// TwinCAT 3 PLC project tc_project_app
// ProgramVersion: 3.1.4022.2
// libraries:
//   Tc2_EtherCAT, * (Beckhoff Automation GmbH)
//   Tc2_MC2, * (Beckhoff Automation GmbH)
//   Tc2_Standard, * (Beckhoff Automation GmbH)
//   Tc2_System, * (Beckhoff Automation GmbH)
//   Tc2_Utilities, * (Beckhoff Automation GmbH)
//   Tc3_Module, * (Beckhoff Automation GmbH)
// project tree:
//   DUTs/ E_MOTION_MODE.TcDUT, E_OPERATION_MODE.TcDUT, E_OPERATION_MODE_NO.TcDUT, E_PHASING_STATE_MACHINE.TcDUT, E_POSITIONING_STATE_MACHINE.TcDUT, E_VELOCITY_STATE_MACHINE.TcDUT (not stored), ST_AXIS_COMMAND.TcDUT, ST_AXIS_STATUS.TcDUT, ST_CMD_EPICS.TcDUT, ST_STAT_EPICS.TcDUT, ST_INDRADRIVE_IO_INPUT.TcDUT (not stored), ST_INDRADRIVE_IO_OUTPUT.TcDUT, ST_S134_MASTERCONTROLWORD.TcDUT, ST_S135_DRIVESTATUSWORD.TcDUT, ST_S144_SIGNALSTATUSWORD.TcDUT (not stored), ST_S145_SIGNALCONTROLWORD.TcDUT (not stored), TARGET_STATE_MACHINE.TcDUT
//   GVLs/ GVL_ErrorCodes.TcGVL, GVL_Parameters.TcGVL
//   / PlcTask.TcTTO
//   POUs/ MAIN_NORMAL_MOTION.TcPOU (not stored), MAIN.TcPOU
//   POUs/Target/ EL3214.TcPOU, fbIndraDrive.TcPOU, FB_BrakeTorque.TcPOU, FB_ModePhasing.TcPOU, FB_ModeVelo.TcPOU, FB_ModePos.TcPOU, FB_ModeHome.TcPOU, FB_PID.TcPOU, FB_RampVelo.TcPOU, FB_PWM.TcPOU, FB_TargetSuperImpose.TcPOU
//   tc_mca_std_lib/DUTs/ DUT_AxisStatus_v0_01.TcDUT (not stored)
//   tc_mca_std_lib/GVLs/ GVL.TcGVL (not stored)
//   tc_mca_std_lib/POUs/ChangeConfig/ FB_ReadFloatParameter.TcPOU (not stored), FB_ReadParameterInNc_v1_00.TcPOU (not stored), FB_WriteFloatParameter.TcPOU (not stored), FB_WriteParameterInNc_v1_00.TcPOU (not stored)
//   tc_mca_std_lib/POUs/ErrorHandling/ DUT_ErrorState.TcDUT (not stored), DUT_TerminalError.TcDUT (not stored), FB_ErrorList.TcPOU (not stored), FB_TerminalError.TcPOU (not stored), GVL_ErrorSystem.TcGVL (not stored), ST_ErrorSystem.TcDUT (not stored)
//   tc_mca_std_lib/POUs/Hardware/EtherCAT_Terminals/Analog_Inputs/ EL3174_0002.TcPOU (not stored), EL3255.TcPOU (not stored), FB_CalculateFrequency_3702_v0_01.TcPOU (not stored)
//   tc_mca_std_lib/POUs/Hardware/EtherCAT_Terminals/Digital_Inputs/ EL1008.TcPOU (not stored), EL1018.TcPOU (not stored), EL1808.TcPOU (not stored), EL1809.TcPOU (not stored), EL1819.TcPOU (not stored), FB_EL1252ASM_v1_00.TcPOU (not stored)
//   tc_mca_std_lib/POUs/Hardware/EtherCAT_Terminals/Digital_Outputs/ EL2014.TcPOU (not stored), EL2252.TcPOU (not stored), EL2808.TcPOU (not stored), EL2819.TcPOU (not stored)
//   tc_mca_std_lib/POUs/Hardware/EtherCAT_Terminals/Digital_Outputs/External_Types/ dutEL2521_Ctrl.TcDUT (not stored), dutEL2521_Status.TcDUT (not stored)
//   tc_mca_std_lib/POUs/Hardware/EtherCAT_Terminals/Measuring_Terminals/ EL5002.TcPOU (not stored), EL5021.TcPOU (not stored), EL5042.TcPOU (not stored), EL5101.TcPOU (not stored)
//   tc_mca_std_lib/POUs/Hardware/EtherCAT_Terminals/Motion/ EL7211_v1_00.TcPOU (not stored), EL9576_v1_00.TcPOU (not stored)
//   tc_mca_std_lib/POUs/Hardware/EtherCAT_Terminals/System/ EL9410.TcPOU (not stored), EL9505.TcPOU (not stored)
//   tc_mca_std_lib/POUs/Hardware/Other/ EK1200.TcPOU (not stored)
//   tc_mca_std_lib/POUs/Motion/ FB_DriveVirtual.TcPOU (not stored), FB_NcAxis.TcPOU (not stored)
//   tc_mca_std_lib/POUs/Motion/Homing/ FB_HomeDirect.TcPOU (not stored), FB_HomeFinish.TcPOU (not stored), FB_HomePrepare.TcPOU (not stored), FB_HomeReadNcVelocities.TcPOU (not stored), FB_HomeReadSoftLimEnable.TcPOU (not stored), FB_HomeToSwitch.TcPOU (not stored), FB_HomeVirtual.TcPOU (not stored), FB_HomeWriteNcVelocities.TcPOU (not stored), FB_HomeWriteSoftLimEnable.TcPOU (not stored)
//   tc_mca_std_lib/VISUs/ FbDriveVisual.TcVIS (not stored), Visualization.TcVIS (not stored)
// (motion and I/O tree: see PLC project tc_epicscommodule)
// real-time tasks:
//   TASK PlcTaskCom: cycle T#1ms, priority 26, ADS port 350
//   TASK PlcTask: cycle T#1ms, priority 20, ADS port 351

CONFIGURATION tc_project_app
    RESOURCE PLC ON TwinCAT3
        TASK PlcTask(INTERVAL := T#1ms, PRIORITY := 20);
        PROGRAM MAIN WITH PlcTask : MAIN;
    END_RESOURCE
END_CONFIGURATION

// ---- DUTs/E_MOTION_MODE.TcDUT
{attribute 'qualified_only'}
{attribute 'strict'}
TYPE E_MOTION_MODE :
(
	eStop 			:= 0, 
	eJogPositive	:= 1, 
	eJogNegative	:= 2, 
	ePositioning 	:= 3 
);
END_TYPE

// ---- DUTs/E_OPERATION_MODE.TcDUT
{attribute 'qualified_only'}
{attribute 'strict'}
TYPE E_OPERATION_MODE :
(
	eTorqueControl										:= 16#0001,
	eVelocityControl									:= 16#0002,
	ePositionControl_Enc1								:= 16#0003,
	ePositionControl_Enc2								:= 16#0004,
	ePositionControl_Lagless_Enc1						:= 16#000B,
	ePositionControl_Lagless_Enc2						:= 16#000C,
	ePositionControl_DriveControlled_Enc1				:= 16#0103,
	ePositionControl_DriveControlled_Enc2				:= 16#0104,
	ePositionControl_Lagless_Enc1_DriveControlled		:= 16#010B,
	ePositionControl_Lagless_Enc2_DriveControlled		:= 16#010C,
	ePositionControl_DriveControlled_w_AxisControlWord	:= 16#0305,
	ePositionControl_w_AxisControlWord					:= 16#0205,
	eDriveInternal_Interpolation_Enc1					:= 16#0113,
	eDriveInternal_Interpolation_Enc2					:= 16#0114,
	eDriveInternal_Interpolation_Lagless_Enc1			:= 16#011B,
	eDriveInternal_Interpolation_Lagless_Enc2			:= 16#011C,
	eDriveInternal_Interpolation_w_AxisControlWord		:= 16#0315,
	eDriveControlled_Positioning_Enc1					:= 16#0123,
	eDriveControlled_Positioning_Enc2					:= 16#0124,
	eDriveControlled_Positioning_Enc1_Lagless			:= 16#012B,
	eDriveControlled_Positioning_Enc2_Lagless			:= 16#012C,
	eDriveControlled_Positioning_w_AxisControlWord		:= 16#0325,
	ePositioning_BlockModeEnc1							:= 16#0133,
	ePositioning_BlockModeEnc2							:= 16#0134,
	ePositioning_BlockModeLagless_Enc1					:= 16#013B,
	ePositioning_BlockModeLagless_Enc2					:= 16#013C,
	ePositioning_BlockMode_w_AxisControlWord			:= 16#0335,
	eCam_Enc1_VirtualMasterAxis							:= 16#8803,
	eCam_Enc2_VirtualMasterAxis							:= 16#8804,
	eCam_Lagless_Enc1_VirtualMaster_Axis				:= 16#880B,
	eCam_Lagless_Enc2_VirtualMaster_Axis				:= 16#880C,
	eCam_Enc1_RealMasterAxis							:= 16#8813,
	eCam_Enc2_RealMasterAxis							:= 16#8814,
	eCam_Lagless_Enc1_RealMasterAxis					:= 16#881B,
	eCam_Lagless_Enc2_RealMasterAxis					:= 16#881C,
	ePhaseSynch_Enc1_VirtualMasterAxis					:= 16#9003,
	ePhaseSynch_Enc2_VirtualMasterAxis					:= 16#9004,
	ePhaseSynch_Lagless_Enc1_VirtualMasterAxis			:= 16#900B,
	ePhaseSynch_Lagless_Enc2_VirtualMasterAxis			:= 16#900C,
	ePhaseSynch_Enc1_RealMasterAxis						:= 16#9013,
	ePhaseSynch_Enc2_RealMasterAxis						:= 16#9014,
	ePhaseSynch_Lagless_Enc1_RealMasterAxis				:= 16#901B,
	ePhaseSynch_Lagless_Enc2_RealMasterAxis				:= 16#901C,
	eVelocitySynch_VirtualMasterAxis					:= 16#A002,
	eVelocitySynch_RealMasterAxis						:= 16#A012,
	eMotionProfileEnc1_VirtualMasterAxis				:= 16#9803,
	eMotionProfileEnc2_VirtualMasterAxis				:= 16#9804,
	eMotionProfile_Lagless_Enc1_VirtualMasterAxis		:= 16#980B,
	eMotionProfile_Lagless_Enc2_VirtualMasterAxis		:= 16#980C,
	eMotionProfileEnc1_RealMasterAxis					:= 16#9813,
	eMotionProfileEnc2_RealMasterAxis					:= 16#9814,
	eMotionProfile_Lagless_Enc1_RealMasterAxis			:= 16#981B,
	eMotionProfile_Lagless_Enc2_RealMasterAxis			:= 16#981C,
	eVelocity_Synch										:= 16#0142,	
	ePosition_Synch										:= 16#0345
) UINT;
END_TYPE

// ---- DUTs/E_OPERATION_MODE_NO.TcDUT
{attribute 'qualified_only'}
{attribute 'strict'}
TYPE E_OPERATION_MODE_NO :
(
	ePrimaryOpMode 		:= 0, 
	eSecondaryOpMode1 	:= 1, 
	eSecondaryOpMode2 	:= 2, 
	eSecondaryOpMode3 	:= 3, 
	eSecondaryOpMode4 	:= 4, 
	eSecondaryOpMode5 	:= 5, 
	eSecondaryOpMode6 	:= 6, 
	eSecondaryOpMode7 	:= 7	
);
END_TYPE

// ---- DUTs/E_PHASING_STATE_MACHINE.TcDUT
{attribute 'qualified_only'}
{attribute 'strict'}
TYPE E_PHASING_STATE_MACHINE :
(
	POWER_OFF := 0,
	POWER_ON :=1,
	ACCELERATION :=2,
	PHASING :=3
);
END_TYPE

// ---- DUTs/E_POSITIONING_STATE_MACHINE.TcDUT
{attribute 'qualified_only'}
{attribute 'strict'}
TYPE E_POSITIONING_STATE_MACHINE :
(
	POWER_OFF := 0,
	POWER_ON := 1,
	POSITION := 2
);
END_TYPE

// ---- DUTs/ST_AXIS_COMMAND.TcDUT
TYPE ST_AXIS_COMMAND :
STRUCT
	eOperationMode				: E_OPERATION_MODE_NO	:= E_OPERATION_MODE_NO.ePrimaryOpMode;	// (S134.0-2) Defines the Operation mode to use (the different operation modes are configured in the drive) 
	bEnableAxis					: BOOL	:= FALSE; 	// FALSE (S134.13-15): Disable drive 
													// TRUE (S134.13-15): Enable drive (torque on the motor) 
	bHaltAxis					: BOOL	:= FALSE;	// FALSE (S134.13-15): Drive performs a HALT operation (Deceleration of drive while maintaining the max. acceleration (S-0-0138). Requires bEnableAxis to be TRUE) 
													// TRUE (S134.13-15): Drive is not halted
	eMotionMode					: E_MOTION_MODE		:= E_MOTION_MODE.eStop;	// Defines the type of motion that shall be performed. This is not functional in Operation Mode Drive internal interpolation! 
	//bPositioningMode			: BOOL;				// (S346.2&1 FALSE&FALSE): Activates positioning mode according to current Operation mode 
	//bJogPositive				: BOOL;				// (S346.2&1 FALSE&TRUE): Activates jogging in positive direction  
	//bJogNeagtive				: BOOL;				// (S346.2&1 TRUE&FALSE): Activates jogging in negative direction
	//bStopAxis					: BOOL;				// (S346.2&1 TRUE&TRUE): Stops the axis 
	bCommandPositionChange		: BOOL	:= FALSE;	// (S346.5) FALSE: Drive moves to current target position, before positioning to new target position (when bCommandValueAccept is toggled) 
													// (S346.5) TRUE: Immediate of target position, i.e., drive immediately acknowledges the new target position (when bCommandValueAccept is toggled) 
	fCommandPosition			: LREAL	:= 0.0;		// (S47, S258 or S282 according to OperationMode)
	fCommandVelocity			: LREAL	:= 0.0; 	// (S259): The velocity used for Positioning and Jogging
	fCommandAcceleration		: LREAL	:= 0.0;		// (S260): The acceleration used for Positioning and Jogging 
	fCommandDeceleration		: LREAL	:= 0.0;		// (S359): The deceleration used for Positioning and Jogging 
	fFeedrateOverride			: LREAL	:= 100.0; 	// (S108):  Parameter used for variable adjustment of the velocity [0..100%] 
	fTorqueLimit				: LREAL	:= 100.0;	// (S92):  Parameter used for limiting the torque [0..drive/motor limit%] 
	bPositionCommandValue		: BOOL	:= FALSE;	// (S346.3): FALSE: Command position is absolute 
													// (S346.3): TRUE: Command position is relative
	bCommandValueAccept			: BOOL	:= FALSE; 	// (S346.0) Toggle bit (FALSE->TRUE or TRUE->FALSE) to start a positioning command in Operation mode "Drive controlled Positioning"
	bCmd_ErrorReset				: BOOL	:= FALSE;	// (S99): Reset the error of the drive 
	bCmd_SetAbsolutePosition	: BOOL	:= FALSE;	// (P12, C0300): Sets the Absolute position of the drive according to drive configuration 
	bCmd_DriveControlledHoming	: BOOL	:= FALSE;	// (S148, C0600): Starts the homing procedure configured in the drive. NOTE that this does not set the absolute position 
	bCmd_DisableLimits			: BOOL	:= FALSE;	// (bS159, C1300): Disables Monitoring of Position error, Position command error, Velocity error and Acceleration limit
	bCmd_ActivateParameterMode	: BOOL	:= FALSE;	//  (S420, C0400): TRUE: Brings the drive to parameter mode 
	bCmd_ExitParameterMode		: BOOL	:= FALSE;	//  (S422, C0200): TRUE: Brings the drive from parameter mode 
	bCmd_RunVirtualMater		: BOOL	:= FALSE;	//  Jog command to the virtual Master
	fVelocityCommandValue		: LREAL	:= 0.0; 	// (S40): The velocity used for Positioning and Jogging

END_STRUCT
END_TYPE

// ---- DUTs/ST_AXIS_STATUS.TcDUT
TYPE ST_AXIS_STATUS :
STRUCT

	bDriveInParameterMode		: BOOL;		// FALSE (S424): Drive is in Operating mode
											// TRUE (S424): The drive is in parameter mode (parameterization level 1 is active)
	eActualOperationModeNo		: E_OPERATION_MODE_NO	:= E_OPERATION_MODE_NO.ePrimaryOpMode;	// (S134.0-2) Defines the Operation mode to use (the different operation modes are configured in the drive) 
	bDCBusPresent				: BOOL;		// FALSE: DC-bus is not present (drive status bb)
											// TRUE (S135.1&0 TRUE&FALSE): DC-bus present (drive state Ab)
	bAxisEnabled				: BOOL; 	// TRUE (S135.1&0 TRUE&TRUE): Axis is operational with torque (drive state AF)
	bAxisHomedStatus			: BOOL; 	// TRUE (S403.0): Axis absolute position is established 
	bAxisStandStillStatus		: BOOL;		// TRUE (S331): Axis is standing still (velocity below configured threshold) 
	bAxisInTargetPosition		: BOOL;		// TRUE (S437.2): Axis command position is reached
	bAxisConstantVelocityStatus	: BOOL;		// TRUE (S437.4): Axis in constant velocity
	bAxisAccelerationStatus		: BOOL;		// TRUE (S437.5): Axis in acceleration
	bAxisDecelerationStatus		: BOOL;		// TRUE (S437.6): Axis in deceleration
	bAxisJogStatus				: BOOL;		// TRUE (S437.12): Axis in jog mode
	fActualPosition				: LREAL;	// The actual position of the axis
	fActualVelocity				: LREAL;	// The actual velocity of the axis
	fActualTorque				: LREAL;	// The actual torque of the axis
	fPositionError				: LREAL;	// The position error of the axis, i.e. the deviation between the Axis Set position and Actual position
	bCommandChange				: BOOL;		// (S135.5): Bit that toggle every time a new command has been recognised by the drive 
	bCommandValueProcessing		: BOOL;		// FALSE (S115.3): Drive ignores (external) command value input (S47, S258, S282 etc) 
											// TRUE (S115.3): Drive follows (external) command value input (S47, S258, S282 etc) 
	bLimitsDisabled				: BOOL;		// TRUE (S159-C1300): 	Monitoring of Position error, Position command error, Velocity error and Acceleration limit is disabled
											// FALSE (S159-C1300): 	Monitoring of Position error, Position command error, Velocity error and Acceleration limit is enabled 
	bDiagMessage				: BOOL;		// TRUE (S135.11): There is a Diagnostic message on the drive 
	bWarning					: BOOL;		// TRUE (S135.12): There is a warning present on the drive 
	bError 						: BOOL;		// TRUE (S135.13): There is an error present on the drive 
	nDiagMessage				: DWORD;	// (S390) Displays the actual diagnostic message on the drive 
END_STRUCT
END_TYPE

// ---- DUTs/ST_CMD_EPICS.TcDUT
TYPE ST_CMD_EPICS :
STRUCT
	
	bExecute:BOOL:=FALSE;
	bEnable:BOOL:=FALSE;
	bReset:BOOL:=FALSE;
	fVelSet:LREAL:=0;
	fPosSet:LREAL:=0;
	eTargetStateCmd: TARGET_STATE_MACHINE:=0;
	
	//brake
	bBrakeLockOnCmd:BOOL:=FALSE;
	bFreeWheelOnOnCmd:BOOL:=TRUE;
	fBrakeSpNm:LREAL:=0;
END_STRUCT
END_TYPE

// ---- DUTs/ST_STAT_EPICS.TcDUT
TYPE ST_STAT_EPICS :
STRUCT
	
	bError:BOOL:=FALSE;
	nErrorId:UDINT:=0;
	bEnabled:BOOL:=FALSE;
	eTargetState: TARGET_STATE_MACHINE;
    sErrorStr:STRING:='NO ERROR';
	fActTorque:LREAL:=0;
	fActPos:LREAL:=0;
	fActVel:LREAL:=0;	
	fActTemp:LREAL:=0;
	fSetVelRaw:LREAL;
	fBrakeActTemp1:LREAL;
	fBrakeActTemp2:LREAL;
	bBrake1TempAlarm:BOOL;
	bBrake2TempAlarm:BOOL;
END_STRUCT
END_TYPE

// ---- DUTs/ST_INDRADRIVE_IO_OUTPUT.TcDUT
TYPE ST_INDRADRIVE_IO_OUTPUT :	// Contains the data that is sent to the drive
STRUCT
	stS134_MasterControlWord			AT %Q*	: ST_S134_MASTERCONTROLWORD; 	
	nS47_PositionCommandValue			AT %Q*	: DINT; 
	nS258_TargetPosition				AT %Q*	: DINT; 
	nS282_PositioningCommandValue		AT %Q*	: DINT; 
	nS259_PositioningVelocity			AT %Q*	: UDINT; 
	nS260_PositioningAcceleration		AT %Q*	: UDINT; 
	nS359_PositioningDeceleration		AT %Q*	: UDINT; 
	nS108_FeedrateOverride				AT %Q*	: UINT; 
	stS145_SignalControlWord			AT %Q*	: ST_S145_SIGNALCONTROLWORD;
	nS92_BiPolarTorqueLimit				AT %Q*	: INT; 
	nS40_VelocityCommandValue			AT %Q*	: DINT; 

END_STRUCT
END_TYPE

// ---- DUTs/ST_S134_MASTERCONTROLWORD.TcDUT
TYPE ST_S134_MASTERCONTROLWORD :
STRUCT
	{attribute 'hide'}
	bS134_0_CtrlInfo_ServiceCh				: BIT;	// 	Control information for service channel
	{attribute 'hide'}
	bS134_1_CtrlInfo_ServiceCh				: BIT;	// 	Control information for service channel
	{attribute 'hide'}
	bS134_2_CtrlInfo_ServiceCh				: BIT;	// 	Control information for service channel
	{attribute 'hide'}
	bS134_3_CtrlInfo_ServiceCh				: BIT;	// 	Control information for service channel
	{attribute 'hide'}
	bS134_4_CtrlInfo_ServiceCh				: BIT;	// 	Control information for service channel
	{attribute 'hide'}
	bS134_5_CtrlInfo_ServiceCh				: BIT;	// 	Control information for service channel
	{attribute 'hide'}
	bS134_6_RealTime_Bit1					: BIT;	// 	Real time bit1
	{attribute 'hide'}
	bS134_7_RealTime_Bit2					: BIT;	// 	Real time bit2
	bS134_CmdOperationMode_Bit0				: BIT;	// 	(bS134_CmdOpMode_B2 | bS134_CmdOpMode_B2 | bS134_CmdOpMode_B0)
													//	000: Primary mode of operation
													// 	001: Secondary operation mode 1
													// 	010: Secondary operation mode 2, etc
	bS134_CmdOperationMode_Bit1				: BIT;	// 	(bS134_CmdOpMode_B2 | bS134_CmdOpMode_B2 | bS134_CmdOpMode_B0)
													//	000: Primary mode of operation
													// 	001: Secondary operation mode 1
													// 	010: Secondary operation mode 2, etc
	bS134_IPOSYNC							: BIT;	// 	Interpolator clock, toggles when new command values are to be transmitted 
	bS134_CmdOperationMode_Bit2				: BIT;	// 	(bS134_CmdOpMode_B2 | bS134_CmdOpMode_B2 | bS134_CmdOpMode_B0)
													//	000: Primary mode of operation
													// 	001: Secondary operation mode 1
													// 	010: Secondary operation mode 2, etc
	{attribute 'hide'}
	bS134_12_Reserved						: BIT;	// 	Reserved
	bS134_DriveHalt							: BIT;	// 	1-0 change: deceleration of drive while maintaining the max. acceleration (S-0-0138) 
													//	(only possible when bit bS134_DriveEnable and bS134_DriveOn = TRUE)
	bS134_DriveEnable						: BIT;	// 	TRUE -> FALSE transition: torque disable without delay (independent of bit bS134_DriveOn or bS134_DriveHalt)
	bS134_DriveOn							: BIT;	// 	TRUE -> FALSE transition: best possible deceleration (only possible if bit bS134_DriveEnable = TRUE)


	

	


END_STRUCT
END_TYPE

// ---- DUTs/ST_S135_DRIVESTATUSWORD.TcDUT
TYPE ST_S135_DRIVESTATUSWORD :
STRUCT
	{attribute 'hide'}
	bS135_0_CtrlInfo_ServiceCh				: BIT;	// 	Control information for service channel
	{attribute 'hide'}
	bS135_1_CtrlInfo_ServiceCh				: BIT;	// 	Control information for service channel
	{attribute 'hide'}
	bS135_2_CtrlInfo_ServiceCh				: BIT;	// 	Control information for service channel
	{attribute 'hide'}
	bS135_3_CmdValProcessingStatus			: BIT;	// 	Status of command value processing
	{attribute 'hide'}
	bS135_4_Reserved						: BIT;	// 	Reserved
	bS135_CommandChange 					: BIT;	// 	Toggling bit to acknowledge that the Command status has changed 
	{attribute 'hide'}
	bS135_6_RealTime_Bit1					: BIT;	// 	Real time bit1
	{attribute 'hide'}
	bS135_7_RealTime_Bit2					: BIT;	// 	Real time bit2
	bS135_ActualOperationMode_Bit0			: BIT;	// 	(bS135_ActOpMode_B2 | bS135_ActOpMode_B2 | bS135_ActOpMode_B0)
													//	000: Primary operation mode active
													// 	001: Secondary operation mode 1 active
													// 	010: Secondary operation mode 2 active, etc
	bS135_ActualOperationMode_Bit1			: BIT;	// 	(bS135_ActOpMode_B2 | bS135_ActOpMode_B2 | bS135_ActOpMode_B0)
													//	000: Primary operation mode active
													// 	001: Secondary operation mode 1 active
													// 	010: Secondary operation mode 2 active, etc
	bS135_ActualOperationMode_Bit2			: BIT;	// 	(bS135_ActOpMode_B2 | bS135_ActOpMode_B2 | bS135_ActOpMode_B0)
													//	000: Primary operation mode active
													// 	001: Secondary operation mode 1 active
													// 	010: Secondary operation mode 2 active, etc
	bS135_Class3_Diag_Mess					: BIT;	// 	TRUE: There is a Class 3 Diagnostic message present in the drive
	bS135_Class2_Diag_Warn					: BIT;	// 	TRUE: There is a Warning present in the drive
	bS135_Class1_Diag_Err					: BIT;	// 	TRUE: There is a Error present in the drive
	bS135_ReadyForOperation_Bit0			: BIT;	// 	(bS135_ReadyForOp_B1 | bS135_ReadyForOp_B0)
													//	00: Not ready for power on (e.g. drive in "P2")
													//	01: Ready for power on ("bb") (A0013)
													//	10: Control section and power section ready for op. ("Ab") (A0012)
													//	11: In operation, with torque (e.g. "AF")
	bS135_ReadyForOperation_Bit1			: BIT;	// 	(bS135_ReadyForOp_B1 | bS135_ReadyForOp_B0)
													//	00: Not ready for power on (e.g. drive in "P2")
													//	01: Ready for power on ("bb") (A0013)
													//	10: Control section and power section ready for op. ("Ab") (A0012)
													//	11: In operation, with torque (e.g. "AF")

	


	


END_STRUCT
END_TYPE

// ---- DUTs/TARGET_STATE_MACHINE.TcDUT
{attribute 'qualified_only'}
{attribute 'strict'}
TYPE TARGET_STATE_MACHINE :
(
	POWER_OFF := 0,
	POWER_ON := 1,
	CONSTANT_VELOCITY :=2,
	POSITIONING :=3,
	PHASING :=4,
	HOMING := 5
	
	
	
);
END_TYPE

// ---- GVLs/GVL_ErrorCodes.TcGVL
{attribute 'qualified_only'}
VAR_GLOBAL
	nErrorCodeOKId:UDINT:=0;
	nErrorCodeOKStr:STRING:='NO ERROR';
	nErrorNoLatchId:UDINT:=1000;
	sErrorNoLatchStr:STRING:='NO LATCH FROM DRIVE';
END_VAR

// ---- GVLs/GVL_Parameters.TcGVL
{attribute 'qualified_only'}
VAR_GLOBAL
	fSpeedToleranceRpm: LREAL := 0.05;
END_VAR

VAR_GLOBAL CONSTANT
	nSectors: LREAL :=36;
    nPulseFreqHz:LREAL:=14;
	fNominalSpeedRpm: LREAL := GVL_Parameters.nPulseFreqHz/GVL_Parameters.nSectors*60;
	fNominalSpeedAdjust: LREAL:=0.001;//-0.0002;  //Timing system vs drive clock tuning. Automize later!
	fPhaseSpeedTol:LREAL:=0.02;   //Speed for last rev needs to be below before start to phase
	fHomeSpeedRpm: LREAL := 1;
    fMaximumSPeedRpm: LREAL := GVL_Parameters.fNominalSpeedRpm*1.1;
	nMaxMotorTemperature: INT:= 80;
	nMaxBrakeTemperature: INT:= 100;
	fWheelDiameter:LREAL:=2500;
	fAccDefault:LREAL:=0.039;  //RPM/S^2 (0.039 => tn min to 23.3) 
	nPhaseErrorFilterSize:INT:=36;  //Two revs
	nVeloInRangeCount:INT:=100;
	nSuperPosMaxCyclesToOutput:INT:=100;
	fSuperPosDutyCycle:LREAL:=2.0/3.0;
	nTaskSampleTime:INT:=1;
	nPhasePIDReducedSampleRateFactor:INT:=1;   //run pid every time new pulse
END_VAR

// ---- POUs/MAIN.TcPOU
PROGRAM MAIN
VAR
	stAmsNetId	AT %I*	              : AMSNETID;
	nPort	AT %I*                    : WORD;
	nMasterAxisPosition AT %I*        : DINT;
	nAdditivePositionSetpoiunt AT %Q* : DINT;
	nAdditiveTorqueSetpoint    AT %Q* : INT;   // Unit 0.1%  (10=1%)
	dLatchedPosition AT %I*           : DINT;
	iBrakeSpRaw AT %Q*                : INT := 0;
	//iRotMotorTempRaw AT %I*           : INT := 0;
    fbTemp                            : EL3214;
	bBrakeFreewheelOn AT %Q*          : BOOL;
	bBrakeLockedOn AT %Q*             : BOOL;
    inputDummy AT %I*                 : BOOL;
	inputDigSens1 AT %I*              : BOOL;
	inputDigSens2 AT %I*              : BOOL;
	fbBrakeTorque                     : FB_BrakeTorque;  // Control brake
	fbModePhase                       : FB_ModePhasing;	 // Phasing Mode
	fbRampVelo                        : FB_RampVelo;
	fbModeVelo                        : FB_ModeVelo;     // Velocity Mode
	fbModePos                         : FB_ModePos;      // Positioning Mode
	fbModeHome                        : FB_ModeHome;     // Homing Mode
	fbIndraDrive                      : fbIndraDrive;    // Control of drive
	stStatEpics                       : ST_STAT_EPICS;   // Status to EPICS
	stCmdEpics                        : ST_CMD_EPICS;    // Control to EPICS 
	stCommands                        : ST_AXIS_COMMAND; // Control to drive
	stStatus                          : ST_AXIS_STATUS;  // Status from drive
	eTargetStateOld                   : TARGET_STATE_MACHINE;
	addStartupTorqueTrigger           : BOOL:=FALSE;
	iTorqueCommandValue  AT %Q*       : INT := 0;
END_VAR

// Monitor temperature
ACT_Temperature();
// Control brake
ACT_Brake();


// Enable Axis independent of state
stCommands.bEnableAxis :=stCmdEpics.bEnable;
stCommands.bHaltAxis:=stCmdEpics.bExecute;
stStatEpics.bEnabled:=stStatus.bAxisEnabled;
stCommands.bCmd_ErrorReset:=stCmdEpics.bReset;

IF NOT stCmdEpics.bEnable THEN
  stCmdEpics.bExecute:=FALSE;
END_IF

stCommands.fCommandAcceleration:=GVL_Parameters.fAccDefault;
stCommands.fCommandDeceleration:=GVL_Parameters.fAccDefault;
stCommands.bCmd_DriveControlledHoming:=FALSE;

// Only allow state change if execute is low
IF stCmdEpics.eTargetStateCmd <> stStatEpics.eTargetState AND NOT stCmdEpics.bexecute THEN
	stStatEpics.eTargetState:=stCmdEpics.eTargetStateCmd;
END_IF

//nAdditiveTorqueSetpoint:=0;
//IF NOT  stCmdEpics.bExecute THEN
//	addStartupTorqueTrigger:=TRUE;
//END_IF

CASE stStatEpics.eTargetState OF 
	TARGET_STATE_MACHINE.CONSTANT_VELOCITY:
		fbModeVelo(
            bExecute:=         stCmdEpics.bExecute,
            bReset:=           stCmdEpics.bReset,
			fVelSet:=          stCmdEpics.fVelSet,
			stStatus:=	       stStatus,	
			stCommands:=       stCommands);
			
			//ramp velocity with selected acceleration
			fbRampVelo(bExecute:=stCmdEpics.bExecute,
              fVelSetIn:=fbModeVelo.fSpeedSetpoint,
              iBlockSampleTimeMicroS:=GVL_Parameters.nTaskSampleTime*1000,
              fVelSetOut:=stCommands.fVelocityCommandValue,
              fVelActIn:=stStatus.fActualVelocity/10);
			  
// add extra torque att startup TEST
		//	IF stStatus.bAxisEnabled AND stCmdEpics.bExecute AND stCmdEpics.fVelSet > 0 THEN
		//		IF stStatus.fActualVelocity/10< stCmdEpics.fVelSet/2 THEN
		//	        nAdditiveTorqueSetpoint:=100;  //Add 10% when under x rpm
		//		ELSIF stStatus.fActualVelocity/10 > stCmdEpics.fVelSet/2 THEN
		//			nAdditiveTorqueSetpoint:=40;
		//		END_IF
		//	END_IF

			
	TARGET_STATE_MACHINE.POSITIONING:
		fbModePos(
            bExecute:=         stCmdEpics.bExecute,
            bReset:=           stCmdEpics.bReset,
			fVelSet:=          stCmdEpics.fVelSet,
			fPosSet:=          stCmdEpics.fPosSet,
			stStatus:=         stStatus,	
			stCommands:=       stCommands);
		
	TARGET_STATE_MACHINE.PHASING:
   		fbModePhase(
			bExecute:=         stCmdEpics.bExecute,
            bReset:=           stCmdEpics.bReset,
			stStatus:=	       stStatus,
			dLatchedPosition:= dLatchedPosition,
			ePhaseType:=stCmdEpics.ePhaseCntrlAlg,
			stCommands:=       stCommands);
			
			//ramp velocity with selected acceleration (as long as not phasing)
			IF NOT fbModePhase.bPhasing THEN
              fbRampVelo(bExecute:=stCmdEpics.bExecute,
                fVelSetIn:=fbModePhase.fSpeedSetpoint,
                iBlockSampleTimeMicroS:=GVL_Parameters.nTaskSampleTime*1000,
                fVelSetOut:=stCommands.fVelocityCommandValue,
                fVelActIn:=fbModePhase.fLastSectorVelocity);
			ELSE // if phasing then take setpoint direct from fbModePhase
			  stCommands.fVelocityCommandValue:=fbModePhase.fSpeedSetpoint;
            END_IF
						
	TARGET_STATE_MACHINE.HOMING:
        fbModeHome( 
            bExecute:=         stCmdEpics.bExecute,
            bReset:=           stCmdEpics.bReset,
			fVelSet:=          stCmdEpics.fVelSet,
			fPosSet:=          stCmdEpics.fPosSet,
			stStatus:=	       stStatus,	
			stCommands:=       stCommands);
			
	TARGET_STATE_MACHINE.TORQUE:
		stCommands.eOperationMode:=E_OPERATION_MODE_NO.eSecondaryOpMode7;
	    stCommands.eMotionMode :=e_Motion_mode.eJogPositive;
	
	  ELSE  // No valid state
		  
		stCmdEpics.bExecute:=FALSE;
        stCmdEpics.bEnable:=FALSE;
		stCommands.fVelocityCommandValue:=0;
		stCommands.fCommandVelocity:=0;
		
END_CASE

IF NOT stCmdEpics.bExecute THEN
	stCommands.fVelocityCommandValue:=0;
END_IF

// TODO: Why I put this here?
stCommands.eMotionMode:=E_MOTION_MODE.eStop;

// Rexroth FB
fbIndraDrive(
	AmsNetId:= stAmsNetId, 
	AdsAddr_Port:= nPort, 
	stAxisCommands:= stCommands, 
	stDriveStatus:= , 
	stAxisStatus=> stStatus, 
	stDriveCommands=> );

// Calculate values for status in EPICS
stStatEpics.fSetVelRaw:= DINT_TO_LREAL(MAIN.fbIndraDrive.stDriveCommands.nS40_VelocityCommandValue)/10000;	
stStatEpics.fActPos:=stStatus.fActualPosition;
stStatEpics.fActTorque:=stStatus.fActualTorque;
stStatEpics.fActVel:=stStatus.fActualVelocity/10;

// Error handling
ACT_Error();

eTargetStateOld:=stStatEpics.eTargetState;

ACTION ACT_Brake:
// Function: Control of brake for simulation of traction
// Use at target test rig
// Author: Anders Sandström 2019

bBrakeFreewheelOn:=stCmdEpics.bFreeWheelOnOnCmd;
bBrakeLockedOn:=stCmdEpics.bBrakeLockOnCmd;

fbBrakeTorque(iTorqueValueinNm:=stCmdEpics.fBrakeSpNm);
iBrakeSpRaw:=fbBrakeTorque.iTorqueScaled;
END_ACTION

ACTION ACT_Diag:
// Function: Some parameters just for debugging
// Note: Do not need to be executed, can be watched online anyway..
// Author: Anders Sandström 2019

	stCommands.bCmd_ActivateParameterMode;//True puts the drive in parameter mode
	stCommands.bCmd_DisableLimits;// True disables monitoring of errors
	stCommands.bCmd_DriveControlledHoming;// True starts homing procedure defined in the drive
	stCommands.bCmd_ErrorReset;
	stCommands.bCmd_ExitParameterMode;
	stCommands.bCmd_RunVirtualMater;// Jog command to the virtual master
	stCommands.bCmd_SetAbsolutePosition;
	stCommands.bCommandPositionChange;// Drive moves to the current target position, when bCommandVAlueAccept toggled, drive moves to the new target position
	stCommands.bCommandValueAccept;// Used in "Drive positioning Mode" to update the target position when toggled
	stCommands.bEnableAxis;
	stCommands.bHaltAxis;// Performs halt on the drive, bEnableaxis has to be TRUE
	stCommands.bPositionCommandValue;//0=Absolute;1=Relative
	stCommands.eMotionMode;
	stCommands.eOperationMode;
	stCommands.fCommandAcceleration;// Acceleration used for positioning and jogging
	stCommands.fCommandDeceleration;// Deceleration used for positioning and jogging
	stCommands.fCommandPosition;
	stCommands.fCommandVelocity;// Velocity used for positioning and jogging
	stCommands.fFeedrateOverride;// Parameter used for adjustment of the velocity (0,100)%
	stCommands.fTorqueLimit;
	stCommands.fVelocityCommandValue;// S40, velocity used for positining and jogging (in velocity mode)
	stStatus.bAxisEnabled;
END_ACTION

ACTION ACT_Error:
// Function: Error handling
// Author: Anders Sandström 2019

IF stStatEpics.eTargetState = TARGET_STATE_MACHINE.PHASING THEN
  IF fbModePhase.bError AND NOT stStatEpics.bError THEN
	  stStatEpics.bError:=fbModePhase.bError;
	  stStatEpics.nErrorId:=fbModePhase.nErrorId;
	  stStatEpics.sErrorStr:=fbModePhase.sErrorStr;
  END_IF
  
ELSIF stStatEpics.eTargetState = TARGET_STATE_MACHINE.CONSTANT_VELOCITY THEN
   IF fbModeVelo.bError AND NOT stStatEpics.bError THEN
	  stStatEpics.bError:=fbModeVelo.bError;
	  stStatEpics.nErrorId:=fbModeVelo.nErrorId;
	  stStatEpics.sErrorStr:=fbModeVelo.sErrorStr;
  END_IF
  
ELSIF stStatEpics.eTargetState = TARGET_STATE_MACHINE.POSITIONING THEN
  IF fbModePos.bError AND NOT stStatEpics.bError THEN
	  stStatEpics.bError:=fbModePos.bError;
	  stStatEpics.nErrorId:=fbModePos.nErrorId;
	  stStatEpics.sErrorStr:=fbModePos.sErrorStr;
  END_IF
  
ELSIF stStatEpics.eTargetState = TARGET_STATE_MACHINE.HOMING THEN
  IF fbModeHome.bError AND NOT stStatEpics.bError THEN
	  stStatEpics.bError:=fbModeHome.bError;
	  stStatEpics.nErrorId:=fbModeHome.nErrorId;
	  stStatEpics.sErrorStr:=fbModeHome.sErrorStr;
  END_IF
  
END_IF


IF stcmdEpics.bReset THEN
	stStatEpics.bError:=FALSE;
	stStatEpics.nErrorId:=GVL_ErrorCodes.nErrorCodeOKId;
	stStatEpics.sErrorStr:=GVL_ErrorCodes.nErrorCodeOKStr;
	stStatEpics.bBrake1TempAlarm:=FALSE;
	stStatEpics.bBrake2TempAlarm:=FALSE;
END_IF
END_ACTION

ACTION ACT_Temperature:
// Function: Monitor tempertures
// Interlock motion on temperatures
// Author: Anders Sandström 2019

fbTemp(En:=TRUE);

IF fbTemp.bError THEN
	stCmdEpics.bExecute:=0;
	stCmdEpics.bEnable:=0;
END_IF

stStatEpics.fActTemp:=fbTemp.iAi_Ch1_Value/10.0;
stStatEpics.fBrakeActTemp1:=fbTemp.iAi_Ch2_Value/10.0;
stStatEpics.fBrakeActTemp2:=fbTemp.iAi_Ch3_Value/10.0;

// Motor Temperature Monitoring Interlock
IF (stStatEpics.fActTemp >= GVL_Parameters.nMaxMotorTemperature)  OR fbTemp.iAi_Ch1_Stat >0 THEN
	stCmdEpics.bEnable:= FALSE;
	stCmdEpics.bExecute:= FALSE;	
END_IF

//Brake temperature monitoring Interlock 1
IF (stStatEpics.fBrakeActTemp1 >= GVL_Parameters.nMaxBrakeTemperature) OR fbTemp.iAi_Ch2_Stat >0 OR stStatEpics.bBrake1TempAlarm THEN
	stCmdEpics.bEnable:= FALSE;
	stCmdEpics.bExecute:= FALSE;		
    stStatEpics.bBrake1TempAlarm:=TRUE; 
END_IF
//Brake temperature monitoring Interlock 2
IF (stStatEpics.fBrakeActTemp2 >= GVL_Parameters.nMaxBrakeTemperature) OR fbTemp.iAi_Ch3_Stat >0 OR stStatEpics.bBrake2TempAlarm THEN
	stCmdEpics.bEnable:= FALSE;
	stCmdEpics.bExecute:= FALSE;		
    stStatEpics.bBrake2TempAlarm:=TRUE; 
END_IF
END_ACTION

END_PROGRAM

// ---- POUs/Target/EL3214.TcPOU
//EL3214 | 4-channel analog input terminal, PT100 (RTD)
FUNCTION_BLOCK EL3214

VAR_INPUT
	En: BOOL;
	iTerminal_ID : INT;
END_VAR

VAR_OUTPUT
	EnO: BOOL;
	iAi_Ch1_Value : INT;
	iAi_Ch2_Value : INT;
	iAi_Ch3_Value : INT;
	iAi_Ch4_Value : INT;
	iAi_Ch1_Stat : BYTE;
	iAi_Ch2_Stat : BYTE;
	iAi_Ch3_Stat : BYTE;
	iAi_Ch4_Stat : BYTE;
	bError: BOOL;
END_VAR

VAR
	//Channels
	AI_RTD_Ch_1_Status	AT %I* : WORD;
	AI_RTD_Ch_1_Value 	AT %I* : INT;
	AI_RTD_Ch_2_Status 	AT %I* : WORD;
	AI_RTD_Ch_2_Value 	AT %I* : INT;
	AI_RTD_Ch_3_Status 	AT %I* : WORD;
	AI_RTD_Ch_3_Value 	AT %I* : INT;
	AI_RTD_Ch_4_Status 	AT %I* : WORD;
	AI_RTD_Ch_4_Value 	AT %I* : INT;
	
	//Terminal status
	WcState_WcState AT %I*: BOOL;
	InfoData_State AT %I*: UINT;
END_VAR

(*
* TODO:
* Status words of the channels
*)

EnO := En;

IF En THEN
	iAi_Ch1_Stat:=WORD_TO_BYTE(AI_RTD_Ch_1_Status);
	iAi_Ch2_Stat:=WORD_TO_BYTE(AI_RTD_Ch_2_Status);
	iAi_Ch3_Stat:=WORD_TO_BYTE(AI_RTD_Ch_3_Status);
	iAi_Ch4_Stat:=WORD_TO_BYTE(AI_RTD_Ch_4_Status);
	
    bError:=WcState_WcState OR NOT (InfoData_State=8);
 
	IF bError = FALSE THEN
		iAi_Ch1_Value := AI_RTD_Ch_1_Value;
		iAi_Ch2_Value := AI_RTD_Ch_2_Value;
		iAi_Ch3_Value := AI_RTD_Ch_3_Value;
		iAi_Ch4_Value := AI_RTD_Ch_4_Value;
	ELSE
		iAi_Ch1_Value := 32768;
		iAi_Ch2_Value := 32768;
		iAi_Ch3_Value := 32768;
		iAi_Ch4_Value := 32768;
	END_IF
END_IF

END_FUNCTION_BLOCK

// ---- POUs/Target/FB_BrakeTorque.TcPOU
FUNCTION_BLOCK FB_BrakeTorque
VAR_INPUT
	iTorqueValueinNm: LREAL;
END_VAR
VAR_OUTPUT
	iTorqueScaled: INT; //Scaled torque value 
END_VAR
VAR
	iTorqueMin:LREAL := 2; // Min brake torque in Nm
	iTorqueMax:LREAL := 200; // Max brake torque in Nm
	iVoltageDecMin:INT := 0; // 0V in decimal representation
	iVoltageDecMax:INT := 32767; //10V in decimal representation
END_VAR

// Function: Interface to brake eon target test rig
// Author: Anders Sandström 2018

IF iTorqueValueinNm >=2 THEN	
  iTorqueScaled := LREAL_TO_INT(((iTorqueValueinNm-iTorqueMin)/(iTorqueMax-iTorqueMin))*(iVoltageDecMax-iVoltageDecMin) + iVoltageDecMin);
ELSE
  iTorqueScaled:=0;
END_IF

END_FUNCTION_BLOCK

// ---- POUs/Target/FB_ModePhasing.TcPOU
FUNCTION_BLOCK FB_ModePhasing
VAR_INPUT
	bExecute:BOOL;
	bReset: BOOL;
	stStatus: ST_AXIS_STATUS;
    dLatchedPosition: DINT;
	fPhaseOffsetDeg: LREAL;
    fPhaseControlKp: LREAL := 0.00001;
	///Ti
	fPhaseControlTn: LREAL := 0;
	///Td
	fPhaseControlTv: LREAL := 0;
	///derviative damping
	fPhaseControlTd: LREAL := 0;
	bPhaseControlReset: BOOL := FALSE;
	
	// for own pid (use kp above)
	fPhaseControlKi: LREAL := 0.0001;
	fPhaseControlKd: LREAL := 0.0001;
	fPhaseControlKff: LREAL := 0.0;
END_VAR
VAR_OUTPUT
	bError: BOOL;
	nErrorId: UDINT;
	sErrorStr: STRING:=GVL_ErrorCodes.nErrorCodeOKStr;
	bPhasing:BOOL;
	fSpeedSetpoint: LREAL;
	fCtrlOutput:LREAL;
END_VAR
VAR_IN_OUT
	stCommands: ST_AXIS_COMMAND;
END_VAR
VAR
	fLatchedPositionOld: LREAL;
	fDistBetweenLastPulses: LREAL;
	fLastSectorVelocity: LREAL;
	fVelocityFromDriveScaled: LREAL;
	fClosestSectorId: LREAL;
	nClosestSectorId: INT;
	fLatchedPosition:LREAL;
	//fbPhasePID: Tc2_Utilities.FB_BasicPID;
	fbPhasePID: FB_PID;
	fPhaseError: LREAL;
	fPhaseErrorFiltered:LREAL;
	fPhaseErrorMM: LREAL:=0;
	dLatchedPositionOld:DINT;
	fPhaseErrorAcc:LREAL;
	ii: INT;
	bTestReset: BOOL;
	bNewTriggPulse:BOOL:=FALSE;
	fArrayFiltVelo: ARRAY[ 0 ..35] OF LREAL;
	fArrayPhaseErrorFilt: ARRAY[ 0 ..99] OF LREAL;
	fArrayPhaseErrorLongTime: ARRAY[ 0 ..99] OF LREAL;
	iFiltVeloArrayIndex:INT:=0;
	fLastSectorVelocityOld:LREAL:=0;
	i:INT:=0;
	fMaxValue:LREAL:=0;
	fMinValue:LREAL:=0;
	fRange:LREAL:=0;
	iRangeOKCounter:INT:=0;
	iRangeOKCounterOld:INT:=0;
	nChoosenSector:INT:=0;
	bPhaseAlgTrigg: BOOL;
	fbPWM: FB_PWM;
	fbSuperImpose:FB_TargetSuperImpose;
	bExecuteSuperImpose: BOOL;
	fPhaseErrorSlope: LREAL;
	iNominalVelCounter:INT:=0;
	fDeltaVelo: LREAL;
	bVeloStable:BOOL:=FALSE;
	timerCheckLatchFreq:TON;
	fNomSpeedSetAdjust: LREAL := 0;
	bTEst: BOOL := FALSE;
	fPidAdd: LREAL := 0;
	fCtrlCycleTime: INT;
	fTn: INT;
END_VAR

// Function: 
// 1. Wait for stable velocity then start "phasing" 
// 2. Choose sector for control
// 3. Calculate phase error (buffer several revs and filter)
// 4. Adjust velo setpoint to minimize phase error
// Author: Anders Sandström 2018

stCommands.fCommandDeceleration:=GVL_Parameters.fAccDefault;	
stCommands.fCommandAcceleration:= GVL_Parameters.fAccDefault;
stCommands.eMotionMode :=e_Motion_mode.eJogPositive;
stCommands.eOperationMode:=e_Operation_mode_no.eSecondaryOpMode2;
fVelocityFromDriveScaled:=stStatus.fActualVelocity/10;
bNewTriggPulse:=FALSE;
bPhasing:=FALSE;
fNomSpeedSetAdjust:=GVL_Parameters.fNominalSpeedRpm + GVL_Parameters.fNominalSpeedAdjust; // Adjust speed setpoint
bPhasing:=bPhaseAlgTrigg;

// Reset alg
IF NOT bExecute OR bPhaseControlReset THEN
 bPhaseAlgTrigg:=FALSE;
END_IF

fLatchedPositionOld:=fLatchedPosition;
fLatchedPosition:=DINT_TO_LREAL(dLatchedPosition)/10000.0;

// New trigger from timing system
IF (fLatchedPosition-fLatchedPositionOld)<>0 THEN
  IF(fLatchedPositionOld>fLatchedPosition) THEN
	fDistBetweenLastPulses:=(360-fLatchedPositionOld+fLatchedPosition);
  ELSE
	fDistBetweenLastPulses:=fLatchedPosition-fLatchedPositionOld;
  END_IF
  bNewTriggPulse:=TRUE;
  fLastSectorVelocity:=fDistBetweenLastPulses*GVL_Parameters.nPulseFreqHz*60/360;
  nClosestSectorId:= LREAL_TO_INT(fLatchedPosition/10);
  
  // Check if stable velocity (close to nominal)	
  iRangeOKCounterOld:=iRangeOKCounter;
  fArrayFiltVelo[iFiltVeloArrayIndex]:=fLastSectorVelocity;
  iFiltVeloArrayIndex:=iFiltVeloArrayIndex+1;
  IF iFiltVeloArrayIndex>35 THEN
	iFiltVeloArrayIndex:=0;
  END_IF
  fLastSectorVelocityOld:=fLastSectorVelocity;
  fMaxValue:=fArrayFiltVelo[0];
  fMinValue:=fArrayFiltVelo[0];
  FOR i:=1 TO 35 BY 1 DO
     IF fArrayFiltVelo[i]> fMaxValue THEN
	   fMaxValue:=fArrayFiltVelo[i];  
     END_IF
     IF fArrayFiltVelo[i]< fMinValue THEN
	   fMinValue:=fArrayFiltVelo[i];  
     END_IF
  END_FOR;
  fRange:=fMaxValue-fMinValue;
  IF fRange < GVL_Parameters.fPhaseSpeedTol AND 
     ABS(fNomSpeedSetAdjust-fMinValue) < GVL_Parameters.fPhaseSpeedTol AND  
     ABS(fNomSpeedSetAdjust-fMaxValue) < GVL_Parameters.fPhaseSpeedTol THEN
	IF iRangeOKCounter <= GVL_Parameters.nVeloInRangeCount THEN
      iRangeOKCounter:=iRangeOKCounter+1;
	END_IF
  ELSE
	iRangeOKCounter:=0; 
  END_IF
  bVeloStable:=iRangeOKCounter >= GVL_Parameters.nVeloInRangeCount;
  IF bVeloStable AND NOT bPhaseAlgTrigg (*AND bTEst*) THEN
    nChoosenSector:=nClosestSectorId-1;
    bPhaseAlgTrigg:=TRUE;
    MEMSET(destAddr:=ADR(fArrayPhaseErrorFilt[0]),0,SIZEOF(fArrayPhaseErrorFilt));
    fPhaseErrorFiltered:=0;
  END_IF
END_IF

//Ensure that pulses arrive from timing system when velocity is above certain limit
timerCheckLatchFreq(IN:=fLatchedPosition = fLatchedPositionOld AND ABS(stStatus.fActualVelocity)>0,PT:=LREAL_TO_TIME(1000/GVL_Parameters.nPulseFreqHz*2));

IF NOT bPhaseAlgTrigg THEN
  fPhaseError:=nClosestSectorId*10-fLatchedPosition;
END_IF

IF bNewTriggPulse THEN
  nChoosenSector:=nChoosenSector+1;
  IF nChoosenSector > 35 THEN
    nChoosenSector:=0;
  END_IF	
END_IF

// Calculate phase error
IF bPhaseAlgTrigg THEN
  fPhaseError:=nChoosenSector*10-fLatchedPosition;
  IF fPhaseError >=180 THEN
	fPhaseError:=360-fPhaseError;
  ELSIF fPhaseError<-180 THEN
	fPhaseError:=fPhaseError+360;
  END_IF
ELSE
  fPhaseError:=nClosestSectorId*10-fLatchedPosition;
END_IF
fPhaseErrorMM:=fPhaseError*GVL_Parameters.fWheelDiameter*pi/360.0; 

//Filter phase error
IF bNewTriggPulse THEN
	MEMMOVE(destAddr:=ADR(fArrayPhaseErrorFilt[1]),srcAddr:=ADR(fArrayPhaseErrorFilt[0]),SIZEOF(LREAL)*(GVL_Parameters.nPhaseErrorFilterSize-1));
	fArrayPhaseErrorFilt[0]:=fPhaseErrorMM;
	fPhaseErrorFiltered:=0;
	FOR ii := 0 TO (GVL_Parameters.nPhaseErrorFilterSize-1) DO
		fPhaseErrorFiltered:=fPhaseErrorFiltered+fArrayPhaseErrorFilt[ii];
	END_FOR
	fPhaseErrorFiltered:=fPhaseErrorFiltered/GVL_Parameters.nPhaseErrorFilterSize;
END_IF

IF NOT fbSuperImpose.bBusy  THEN
  bExecuteSuperImpose:= NOT bExecuteSuperImpose;
END_IF

//Drops very fast from positive to negative error. So, Adjust more gently when phase error is positive
IF(fPhaseErrorFiltered > 0) THEN  //Pos error
  IF ABS(fPhaseErrorFiltered)>10 THEN
    fDeltaVelo:= 0.003;
  ELSIF ABS(fPhaseErrorFiltered)>4 THEN
    fDeltaVelo:= 0.0025;
  ELSIF ABS(fPhaseErrorFiltered)>1 THEN
    fDeltaVelo:= 0.002;
  ELSIF ABS(fPhaseErrorFiltered)>0.5 THEN
    fDeltaVelo:= 0.0015;
  ELSE
	fDeltaVelo:= 0.0015;
  END_IF
ELSE // neg error
  IF ABS(fPhaseErrorFiltered)>10 THEN  
    fDeltaVelo:= 0.003;
  ELSIF ABS(fPhaseErrorFiltered)>4 THEN
    fDeltaVelo:= 0.0025;
  ELSIF ABS(fPhaseErrorFiltered)>1 THEN
    fDeltaVelo:= 0.002;
  ELSIF ABS(fPhaseErrorFiltered)>0.5 THEN
    fDeltaVelo:= 0.0015;
  ELSE
	fDeltaVelo:= 0.0015;
  END_IF	
END_IF

//Adjust nominal speed (this function should be automated (adaptive))
fSpeedSetpoint:=fNomSpeedSetAdjust;
IF fSpeedSetpoint>GVL_Parameters.fMaximumSPeedRpm THEN
  fSpeedSetpoint:=GVL_Parameters.fMaximumSPeedRpm; 
END_IF
IF NOT bExecute THEN
  fSpeedSetpoint:=0;	
END_IF
IF bNewTriggPulse AND bPhaseAlgTrigg THEN
 (* fbPhasePID(fSetpointValue:=0,
             fActualValue:=fPhaseErrorFiltered,
             bReset:=bPhaseControlReset,
             fCtrlCycleTime:=0.071,
             fKp:=fPhaseControlKp,
             fTn:=fPhaseControlTn,
             fTv:=fPhaseControlTv,
             fTd:=fPhaseControlTd);*)
  fbPhasePID(fSetpointValue:=0,
             fActualValue := fPhaseErrorFiltered,
             bReset       := bPhaseControlReset,
			 fFF          := 0,
			 fKp          := fPhaseControlKp,
			 fKi          := fPhaseControlKi,
			 fKd          := fPhaseControlKd,
			 fKff         := fPhaseControlKff,
			 fIOutputMin  :=-fDeltaVelo,
			 fIOutputMax  := fDeltaVelo,
			 );
  fPidAdd:=fbPhasePID.fCtrlOutput;
(*  IF ABS(fbPhasePID.fCtrlOutput)>fDeltaVelo THEN
    IF fbPhasePID.fCtrlOutput < 0 THEN
		fPidAdd:=-fDeltaVelo;
	ELSE
		fPidAdd:=fDeltaVelo;	
    END_IF	 
  END_IF*)
ELSIF NOT bPhaseAlgTrigg THEN
  fbPhasePID(bReset:=TRUE);
  fPidAdd:=0;
END_IF

fbSuperImpose(bExecute:=bExecuteSuperImpose AND bPhaseAlgTrigg,
      iSampleRateMs:=GVL_Parameters.nTaskSampleTime,
      fNominalVelocityRpm:=fSpeedSetpoint,
      fMaxDeltaVelocityRpm:=fDeltaVelo,
      fPhaseErrorDeg:=fPhaseErrorFiltered/(GVL_Parameters.fWheelDiameter*pi)*360);  

(*IF fPhaseErrorFiltered < 0 THEN
  fSpeedSetpoint:=fSpeedSetpoint-fDeltaVelo;
ELSE
  fSpeedSetpoint:=fSpeedSetpoint+fDeltaVelo;
END_IF
fbPWM(
       En:=TRUE,
       bEnable:=TRUE,
       iBlockSampleTimeMicroS:=GVL_Parameters.nTaskSampleTime*1000,
       iProcessSampleTimeMicroS:=71000,
       iDecimalPoint:=3,
       fInput:=fSpeedSetpoint);*)

fbPWM(
       En:=TRUE,
       bEnable:=TRUE,
       iBlockSampleTimeMicroS:=GVL_Parameters.nTaskSampleTime*1000,
       iProcessSampleTimeMicroS:=71000,
       iDecimalPoint:=3,
       fInput:=fSpeedSetpoint+fPidAdd);
(*fbPWM(
       En:=TRUE,
       bEnable:=TRUE,
       iBlockSampleTimeMicroS:=GVL_Parameters.nTaskSampleTime*1000,
       iProcessSampleTimeMicroS:=71000,
       iDecimalPoint:=3,
       fInput:=fbSuperImpose.fVelocitySetpointRpm);
	   *)
(*fbPWM(
       En:=TRUE,
       bEnable:=TRUE,
       iBlockSampleTimeMicroS:=GVL_Parameters.nTaskSampleTime*1000,
       iOverrideSampleTimeMicroS:=71000,
       iDecimalPoint:=3,
       fOverrideInput:=fNomSpeedSetAdjust);*)
//stCommands.fVelocityCommandValue:=fbPWM.fOverrideOutput;	
fSpeedSetpoint:=fbPWM.fOutput;
//fSpeedSetpoint:=fbSuperImpose.fVelocitySetpointRpm;
//fSpeedSetpoint:=fNomSpeedSetAdjust;
dLatchedPositionOld:=dLatchedPosition;
 
//*********Errorhandling

// Latched pulses missing
IF timerCheckLatchFreq.Q THEN
	bError:=TRUE;
	nErrorId:=GVL_ErrorCodes.nErrorNoLatchId;
	sErrorStr:=GVL_ErrorCodes.sErrorNoLatchStr;
END_IF

IF bReset THEN
	bError:=FALSE;
	nErrorId:=0;
END_IF

END_FUNCTION_BLOCK

// ---- POUs/Target/FB_PID.TcPOU
FUNCTION_BLOCK FB_PID
VAR_INPUT
	fSetpointValue: LREAL:=0;
	fActualValue :LREAL :=0;
	fFF:LREAL:=0;
	//iBlockSampleTimeMicroS: DINT;
	fKp: LREAL:=0;
	fKi: LREAL:=0;
	fKd: LREAL:=0;
	fKff: LREAL:=0;
	fIOutputMin: LREAL:=0;
	fIOutputMax: LREAL:=0;
	bReset:BOOL:=FALSE;
END_VAR
VAR_OUTPUT
	fCtrlOutput: LREAL;
END_VAR
VAR
	fOutputFF:LREAL:=0;
    fOutputP:LREAL:=0;
	fOutputI:LREAL:=0;
	fOutputD:LREAL:=0;
	fError:LREAL:=0;
	fErrorOld:LREAL:=0;
END_VAR

// Function: Simple PID controller with FF and limits for integral..
// Custom implementation needed since integral high and low limits are 
// needed in order to prvent integral windup.
// Author: Anders Sandström 20200115
 
IF bReset THEN
  fOutputP:=0;
  fOutputI:=0;
  fOutputD:=0;
  fFF:=0;
  fCtrlOutput:=0;
  RETURN;
END_IF

fErrorOld := fError;
fError    := fActualValue-fSetpointValue;

fOutputFF := fFF*fKff;         
fOutputP  := fKp*fError;
fOutputI  := fOutputI + fKi* fError;
// Prevent integral windup
IF fOutputI > fIOutputMax THEN
  fOutputI := fIOutputMax;
ELSIF fOutputI < fIOutputMin THEN
  fOutputI := fIOutputMin; 
END_IF

fOutputD  :=  (fError-fErrorOld)*fKd;

fCtrlOutput := fOutputP + fOutputI + fOutputD + fOutputFF;

END_FUNCTION_BLOCK

// ---- POUs/Target/FB_PWM.TcPOU
FUNCTION_BLOCK FB_PWM
VAR_INPUT
	En: BOOL;
	bEnable: BOOL;
	iBlockSampleTimeMicroS: DINT;
	iProcessSampleTimeMicroS: DINT;
	iDecimalPoint: INT;
	fInput: LREAL;
	//iTrigger:INT:=0;
END_VAR
VAR_OUTPUT
	EnO: BOOL;
	fOutput: LREAL;
END_VAR
VAR
	iNumCycles: DINT;
	iBase: DINT;
	fDecimals: LREAL;
	i: INT;
	iDecimalGain: DINT;
	fOutputHigh: LREAL;
	iHighCycles: DINT;
	iLowCycles: DINT;
	fOutputLow: LREAL;
	iCycleCounter: DINT;
	iLowCounter: INT;
	iHighCounter: INT;
	fActualPWM: LREAL;
	fSetpointPWM: LREAL;
	fOverrideOld: LREAL;
END_VAR


IF bEnable THEN
  //IF(iTrigger<>iTriggerOld) THEN // New fOverride value
    iNumCycles:=iProcessSampleTimeMicroS/iBlockSampleTimeMicroS; //71 if 71ms and 1ms
	iDecimalGain:=1;
	FOR i:=1 TO iDecimalPoint DO
	  iDecimalGain:=iDecimalGain*10; //10000 if iDecimalpoint is 4
	END_FOR
	iBase:=TRUNC(fInput*iDecimalGain); //=900004 if fOverride=90.00045
    fDecimals:=fInput*iDecimalGain-iBase; //=0.5 if fOverride=90.00045
    iHighCycles:=TRUNC(iNumCycles*fDecimals);
    iLowCycles:=iNumCycles-iHighCycles;
    fOutputLow:=DINT_TO_LREAL(iBase)/iDecimalGain; //90.0004
    fOutputHigh:=DINT_TO_LREAL(iBase+1)/iDecimalGain; //90.0005
    //iCycleCounter:=0;
    //iLowCounter:=0;
    //iHighCounter:=0;	
  //END_IF
	
  (*IF ABS(fInput-fOverrideOld)>0 THEN 
	iCycleCounter:=0;
	iLowCounter:=0;
	iHighCounter:=0;	
	fOverrideOld:=fInput;
   END_IF*)

  IF iCycleCounter> iNumCycles THEN
	iCycleCounter:=0;
	iLowCounter:=0;
	iHighCounter:=0;	
  END_IF
  
  iCycleCounter:=iCycleCounter+1;
  IF iLowCycles > 0 THEN
	IF iHighCycles > 0 THEN
	  //Both high and low should be output during the period
	  IF iLowCounter = 0 THEN
		fOutput:=fOutputLow;
		iLowCounter:=iLowCounter+1;
	  ELSE
	    IF iHighCounter = 0 THEN
		  fOutput:=fOutputHigh;
		  iHighCounter:=iHighCounter+1;
	    ELSE //both counters is atleast 1
		  fActualPWM:= DINT_TO_LREAL(iHighCounter)/DINT_TO_LREAL(iLowCounter+iHighCounter);
		  fSetpointPWM:=DINT_TO_LREAL(iHighCycles)/DINT_TO_LREAL(iLowCycles+iHighCycles);
		  IF fActualPWM>fSetpointPWM THEN
		    fOutput:=fOutputLow;
		    iLowCounter:=iLowCounter+1;
		  ELSE
            fOutput:=fOutputHigh;
		    iHighCounter:=iHighCounter+1;
		  END_IF				
	    END_IF				
	  END_IF
    ELSE		
	  fOutput:=fOutputLow;
	  iLowCounter:=iLowCounter+1;
    END_IF
  ELSE
    fOutput:=fOutputHigh;
	iHighCounter:=iHighCounter+1;
  END_IF
ELSE	
	fOutput:=fInput;	
END_IF

END_FUNCTION_BLOCK

// ---- POUs/Target/FB_TargetSuperImpose.TcPOU
FUNCTION_BLOCK FB_TargetSuperImpose
VAR_INPUT
  En: BOOL;
  bExecute: BOOL;
  iSampleRateMs:INT;
  iProcessSampleRateMs:INT:=0;
  fNominalVelocityRpm: LREAL;
  fMaxDeltaVelocityRpm: LREAL;
  fPhaseErrorDeg: LREAL;	
END_VAR
VAR_OUTPUT
	fVelocitySetpointRpm: LREAL;
	bBusy: BOOL;
END_VAR
VAR
	fbRtrig: R_TRIG;
	iCyclesToOutput: INT;
	iCycleCounter: INT;
END_VAR


// Function: Superimpose of positioning (ONLY FOR TARGET)
// Author: Anders Sandström 2018

IF NOT bExecute THEN
	bBusy:=FALSE;
	iCycleCounter:=0;
	iCyclesToOutput:=0;
END_IF

fbRtrig(clk:=bExecute);
IF fbRtrig.Q THEN
  // Calculate new velocity to output
  
  iCyclesToOutput:=LREAL_TO_INT(ABS(fPhaseErrorDeg)/(ABS(fMaxDeltaVelocityRpm)*360.0/60.0)*1000.0/iSampleRateMs*2.0/100.0);
  IF(iCyclesToOutput>GVL_Parameters.nSuperPosMaxCyclesToOutput) THEN
    iCyclesToOutput:=GVL_Parameters.nSuperPosMaxCyclesToOutput;
  END_IF 
END_IF

IF iCycleCounter<iCyclesToOutput*GVL_Parameters.fSuperPosDutyCycle AND bExecute  THEN
  IF fPhaseErrorDeg >= 0 THEN
    fVelocitySetpointRpm:=fNominalVelocityRpm + fMaxDeltaVelocityRpm;
  ELSE 
    fVelocitySetpointRpm:=fNominalVelocityRpm - fMaxDeltaVelocityRpm;
  END_IF
  bBusy:=TRUE;
ELSE
  bBusy:=TRUE;		
  fVelocitySetpointRpm:=fNominalVelocityRpm;
END_IF

IF iCycleCounter<iCyclesToOutput THEN
  iCycleCounter:=iCycleCounter+1;
ELSE
  bBusy:=FALSE;
END_IF

END_FUNCTION_BLOCK

// ---- POUs/Target/FB_RampVelo.TcPOU
FUNCTION_BLOCK FB_RampVelo
VAR_INPUT
	bExecute:BOOL;
	fVelSetIn:LREAL:=0;
	iBlockSampleTimeMicroS:INT:=10000;
	fVelActIn:LREAL:=0;
END_VAR
VAR_IN_OUT
    fVelSetOut:LREAL:=0;
END_VAR
VAR
  fChangePerCycle:LREAL:=0;
  fCurrAcc:LREAL:=0;
  fAccX1:LREAL:=0.8;
  fAccX2:LREAL:=0.99;
  fAccY1:LREAL:=GVL_Parameters.fAccDefault;
  fAccY2:LREAL:=GVL_Parameters.fAccDefault*0.1;
  fAccK:LREAL:=0;
  fAccM:LREAL:=0;
  x:LREAL:=0;
  bExecuteOld:BOOL:=FALSE;
  fActVeloOld:LREAL:=0;  // Used for extra sanity check of velo
END_VAR

// Function: Ramp velocity with a defined acceleration.
// Accelerartion is ramped down when apparching velosity setpoint in order to reduce
// overshoot and oscillations..
// Author: Anders Sandström 20200114

IF NOT bExecute OR fVelSetIn > GVL_Parameters.fMaximumSPeedRpm THEN
  fVelSetOut:=0;
  bExecuteOld:=bExecute;
  RETURN;
END_IF;

// Start at current velocity if retreigger (avoid go to zero)
IF NOT bExecuteOld AND bExecute THEN
  // Sanity check of the actual velocity
  IF fVelActIn > -GVL_Parameters.fMaximumSPeedRpm AND 
	 fVelActIn < GVL_Parameters.fMaximumSPeedRpm AND 
	 fActVeloOld > -GVL_Parameters.fMaximumSPeedRpm AND 
	 fActVeloOld < GVL_Parameters.fMaximumSPeedRpm THEN
	fVelSetOut:=(fVelActIn+fActVeloOld)/2;  //Set to average of two cycles
  ELSE
    fVelSetOut:=0;
  END_IF  
END_IF
bExecuteOld:=bExecute;
fActVeloOld:=fVelActIn;

IF fVelSetOut=fVelSetIn THEN
  fVelSetOut:=fVelSetIn;
  RETURN;
END_IF;

//Reduce overshoot by lowering acc when closing in on setpoint (linear)
//           Acceleration [rpm/s^2]
//                 ^
//  y1=defAcc     -|-----------------\
//                 |                  \  
//                 |                   \
//                 |                    \ 
//                 |                     \
//  y2=defAcc*0.1 -|                      \-----------------
//                 |--------------------------------------------> fSetOut/fSetIn []
//                                 x1=0.8 x2=1.0 
fAccK:=(fAccY2-fAccY1)/(fAccX2-fAccX1);
fAccM:= fAccY1-fAccK*fAccX1;
x:=fVelSetOut/fVelSetIn;
// try linear ramp down off acceleration from 0.8*velsetin to velset in (from defacc to 0.1* defacc)
fCurrAcc:=GVL_Parameters.fAccDefault;
IF x > fAccX1 AND x <= fAccX2 AND fVelSetOut<fVelSetIn THEN
  fCurrAcc:=fAccK*fVelSetOut/fVelSetIn+fAccM;
ELSIF x >= fAccX2 THEN
  fCurrAcc:=GVL_Parameters.fAccDefault*0.1;
END_IF

// Change per execution
fChangePerCycle:=fCurrAcc/(1E6/iBlockSampleTimeMicroS);

// Ramp finished
IF ABS(fVelSetIn-fVelSetOut)<fChangePerCycle THEN
  fVelSetOut:=fVelSetIn;
  RETURN;
END_IF

//Acc
IF fVelSetIn > fVelSetOut THEN             // Acc
  fVelSetOut:=fVelSetOut+fChangePerCycle;
ELSIF fVelSetIn < fVelSetOut THEN          // Dec
  fVelSetOut:=fVelSetOut-fChangePerCycle;
END_IF

END_FUNCTION_BLOCK

// ---- POUs/Target/FB_ModeVelo.TcPOU
FUNCTION_BLOCK FB_ModeVelo
VAR_INPUT
	bExecute:BOOL;
	bReset: BOOL;
	fVelSet:LREAL:=0;
	stStatus: ST_AXIS_STATUS;
END_VAR
VAR_OUTPUT
	fSpeedSetpoint:LREAL:=0;
	bError: BOOL;
	nErrorId: UDINT;
	sErrorStr: STRING:=GVL_ErrorCodes.nErrorCodeOKStr;
END_VAR
VAR_IN_OUT
	stCommands: ST_AXIS_COMMAND;
END_VAR
VAR

END_VAR

// Function: Constant velocity of target main  motor
// Control will be performed by the drive.
// Author: Anders Sandström 2018

stCommands.eMotionMode :=e_Motion_mode.eJogPositive;
stCommands.eOperationMode:=e_Operation_mode_no.eSecondaryOpMode2;
IF bExecute THEN
	fSpeedSetpoint:=fVelSet;
ELSE
	fSpeedSetpoint:=0;
END_IF
stCommands.fCommandVelocity:=0; // Other mode

END_FUNCTION_BLOCK

// ---- POUs/Target/FB_ModePos.TcPOU
FUNCTION_BLOCK FB_ModePos
VAR_INPUT
	bExecute:BOOL;
	bReset: BOOL;
	fVelSet:LREAL:=0;
	fPosSet:LREAL:=0;
	stStatus: ST_AXIS_STATUS;
END_VAR
VAR_OUTPUT
	bError: BOOL;
	nErrorId: UDINT;
	sErrorStr: STRING:=GVL_ErrorCodes.nErrorCodeOKStr;
END_VAR
VAR_IN_OUT
	stCommands: ST_AXIS_COMMAND;
END_VAR
VAR

END_VAR

// Actually not neccesarry to use FB here but nice to keep structure
stCommands.eMotionMode :=e_Motion_mode.ePositioning;
stCommands.eOperationMode:=e_Operation_mode_no.eSecondaryOpMode1;
IF bExecute THEN
  stCommands.fVelocityCommandValue:=fVelSet;
ELSE
  stCommands.fVelocityCommandValue:=0;
END_IF
stCommands.fCommandVelocity:=0;
stCommands.fCommandPosition:=fPosSet;

END_FUNCTION_BLOCK

// ---- POUs/Target/FB_ModeHome.TcPOU
FUNCTION_BLOCK FB_ModeHome
VAR_INPUT
	bExecute:BOOL;
	bReset: BOOL;
	fVelSet:LREAL:=0;
	fPosSet:LREAL:=0;
	stStatus: ST_AXIS_STATUS;
END_VAR
VAR_OUTPUT
	bError: BOOL;
	nErrorId: UDINT;
	sErrorStr: STRING:=GVL_ErrorCodes.nErrorCodeOKStr;
END_VAR
VAR_IN_OUT
	stCommands: ST_AXIS_COMMAND;
END_VAR
VAR

END_VAR

// Function: Initiate homing of target main  motor
// Actual homing will be performed by the drive.
// Author: Anders Sandström 2018

stCommands.eMotionMode:=e_Motion_mode.ePositioning;
stCommands.bCmd_DriveControlledHoming:=bExecute;
stCommands.fVelocityCommandValue:=GVL_Parameters.fHomeSpeedRpm;
stCommands.fCommandVelocity:=GVL_Parameters.fHomeSpeedRpm;

END_FUNCTION_BLOCK

// ---- POUs/Target/fbIndraDrive.TcPOU
FUNCTION_BLOCK fbIndraDrive
VAR_INPUT 
	AmsNetId			: AMSNETID;		// AMS Net Id of the EtherCAT Master
	AdsAddr_Port		: WORD; 		// EtherCAT address of the Drive
	stAxisCommands		: ST_AXIS_COMMAND; 
	stDriveStatus		: ST_INDRADRIVE_IO_INPUT; 
END_VAR
VAR_OUTPUT
	stAxisStatus		: ST_AXIS_STATUS; 
	stDriveCommands		: ST_INDRADRIVE_IO_OUTPUT; 
END_VAR
VAR
	sAmsNetId						: T_AmsNetId;
	fbReadParameter					: FB_EcSoERead;
	nS149_DataStatus				: UDINT	:= 0;
	bDummy: BOOL;
	ii: INT;
END_VAR

VAR CONSTANT
	cC1300_LimitsEnabled			: UDINT := 0;
	cC1300_LimitsDisableActivated	: UDINT := 7;
	cC1300_LimitsDisabled			: UDINT := 3;
END_VAR

//==================================================================================================
//====== FunctionBlock to manage IndraDrive status and command =====================================
//==================================================================================================

// Create the T_AmsNetId 
sAmsNetId := F_CreateAmsNetId(AmsNetId); 

(*==================================================================================================================================================
=============    STATUS FROM THE DRIVE    ==========================================================================================================
==================================================================================================================================================*)
	// Display Drive status
		// Drive parameter mode  
		stAxisStatus.bDriveInParameterMode			:= stDriveStatus.stS144_SignalStatusWord.bS424_DriveMode; 

		// Drive Operation mode number
		IF (NOT stDriveStatus.nS135_DriveStatusWord.bS135_ActualOperationMode_Bit2) AND (NOT stDriveStatus.nS135_DriveStatusWord.bS135_ActualOperationMode_Bit1) AND (NOT stDriveStatus.nS135_DriveStatusWord.bS135_ActualOperationMode_Bit0) THEN 
			stAxisStatus.eActualOperationModeNo	:= E_OPERATION_MODE_NO.ePrimaryOpMode; 
		ELSIF (NOT stDriveStatus.nS135_DriveStatusWord.bS135_ActualOperationMode_Bit2) AND (NOT stDriveStatus.nS135_DriveStatusWord.bS135_ActualOperationMode_Bit1) AND stDriveStatus.nS135_DriveStatusWord.bS135_ActualOperationMode_Bit0 THEN 
			stAxisStatus.eActualOperationModeNo	:= E_OPERATION_MODE_NO.eSecondaryOpMode1; 
		ELSIF (NOT stDriveStatus.nS135_DriveStatusWord.bS135_ActualOperationMode_Bit2) AND stDriveStatus.nS135_DriveStatusWord.bS135_ActualOperationMode_Bit1 AND (NOT stDriveStatus.nS135_DriveStatusWord.bS135_ActualOperationMode_Bit0) THEN 
			stAxisStatus.eActualOperationModeNo	:= E_OPERATION_MODE_NO.eSecondaryOpMode2; 
		ELSIF (NOT stDriveStatus.nS135_DriveStatusWord.bS135_ActualOperationMode_Bit2) AND stDriveStatus.nS135_DriveStatusWord.bS135_ActualOperationMode_Bit1 AND stDriveStatus.nS135_DriveStatusWord.bS135_ActualOperationMode_Bit0 THEN 
			stAxisStatus.eActualOperationModeNo	:= E_OPERATION_MODE_NO.eSecondaryOpMode3; 
		ELSIF stDriveStatus.nS135_DriveStatusWord.bS135_ActualOperationMode_Bit2 AND (NOT stDriveStatus.nS135_DriveStatusWord.bS135_ActualOperationMode_Bit1) AND (NOT stDriveStatus.nS135_DriveStatusWord.bS135_ActualOperationMode_Bit0) THEN 
			stAxisStatus.eActualOperationModeNo	:= E_OPERATION_MODE_NO.eSecondaryOpMode4; 
		ELSIF stDriveStatus.nS135_DriveStatusWord.bS135_ActualOperationMode_Bit2 AND (NOT stDriveStatus.nS135_DriveStatusWord.bS135_ActualOperationMode_Bit1) AND stDriveStatus.nS135_DriveStatusWord.bS135_ActualOperationMode_Bit0 THEN 
			stAxisStatus.eActualOperationModeNo	:= E_OPERATION_MODE_NO.eSecondaryOpMode5; 
		ELSIF stDriveStatus.nS135_DriveStatusWord.bS135_ActualOperationMode_Bit2 AND stDriveStatus.nS135_DriveStatusWord.bS135_ActualOperationMode_Bit1 AND (NOT stDriveStatus.nS135_DriveStatusWord.bS135_ActualOperationMode_Bit0) THEN 
			stAxisStatus.eActualOperationModeNo	:= E_OPERATION_MODE_NO.eSecondaryOpMode6; 
		ELSIF stDriveStatus.nS135_DriveStatusWord.bS135_ActualOperationMode_Bit2 AND stDriveStatus.nS135_DriveStatusWord.bS135_ActualOperationMode_Bit1 AND stDriveStatus.nS135_DriveStatusWord.bS135_ActualOperationMode_Bit0 THEN 
			stAxisStatus.eActualOperationModeNo	:= E_OPERATION_MODE_NO.eSecondaryOpMode7; 
		END_IF
		// DC Bus
		stAxisStatus.bDCBusPresent					:= (*(NOT stDriveStatus.nS135_DriveStatusWord.bS135_ReadyForOperation_Bit0) AND *) stDriveStatus.nS135_DriveStatusWord.bS135_ReadyForOperation_Bit1; 
		// Axis enabled 
		stAxisStatus.bAxisEnabled					:= stDriveStatus.nS135_DriveStatusWord.bS135_ReadyForOperation_Bit0 AND stDriveStatus.nS135_DriveStatusWord.bS135_ReadyForOperation_Bit1; 
		// Absolute position status
		stAxisStatus.bAxisHomedStatus				:= stDriveStatus.stS144_SignalStatusWord.bS403_0_AxisHomedStatus; 
		// Axis standstill status 
		stAxisStatus.bAxisStandStillStatus			:= stDriveStatus.stS144_SignalStatusWord.bS331_StandStillStatus; 
		// Axis in target position
		stAxisStatus.bAxisInTargetPosition			:= stDriveStatus.stS144_SignalStatusWord.bS437_2_CommandPositionReached;
 		// Axis in constant velocity
		stAxisStatus.bAxisConstantVelocityStatus	:= (NOT stDriveStatus.stS144_SignalStatusWord.bS331_StandStillStatus) AND (NOT stDriveStatus.stS144_SignalStatusWord.bS437_5_Acceleration) AND (NOT stDriveStatus.stS144_SignalStatusWord.bS437_6_Deceleration);
 		// Axis in Acceleration
		stAxisStatus.bAxisAccelerationStatus		:= stDriveStatus.stS144_SignalStatusWord.bS437_5_Acceleration;
 		// Axis in Deceleration
		stAxisStatus.bAxisDecelerationStatus		:= stDriveStatus.stS144_SignalStatusWord.bS437_6_Deceleration;
 		// Axis in Jog
		stAxisStatus.bAxisJogStatus					:= stDriveStatus.stS144_SignalStatusWord.bS437_12_JogMode;
		// Drive command change 
		stAxisStatus.bCommandChange					:= stDriveStatus.nS135_DriveStatusWord.bS135_CommandChange; 
		// Drive command value processing  
		stAxisStatus.bCommandValueProcessing		:= stDriveStatus.stS144_SignalStatusWord.bP115_3_StatusOfCmdValueProcessing; 
		
		// Disable monitoring  
		IF 	(stAxisCommands.bCmd_DisableLimits AND (NOT stAxisStatus.bLimitsDisabled)) OR 
			((NOT stAxisCommands.bCmd_DisableLimits) AND stAxisStatus.bLimitsDisabled) THEN
				fbReadParameter(
					sNetId:= sAmsNetId, 
					nSlaveAddr:= AdsAddr_Port, 
					nIdn:= 149, 
					nElement:= 16#01, 
					nDriveNo:= 0, 
					bCommand:= FALSE, 
					pDstBuf:= ADR(nS149_DataStatus), 
					cbBufLen:= SIZEOF(nS149_DataStatus), 
					bExecute:= TRUE, 
					tTimeout:= , 
					bBusy=> , 
					bError=> , 
					nErrId=> ); 
				
				IF (NOT fbReadParameter.bBusy) AND (NOT fbReadParameter.bError) THEN 
					IF (nS149_DataStatus = cC1300_LimitsDisableActivated) OR (nS149_DataStatus = cC1300_LimitsDisabled) THEN 
						stAxisStatus.bLimitsDisabled	:= TRUE;
					ELSIF (nS149_DataStatus = cC1300_LimitsEnabled) THEN 
						stAxisStatus.bLimitsDisabled	:= FALSE;
					END_IF
					// Execute with FALSE
					fbReadParameter(bExecute:= FALSE);
				END_IF
				
				IF fbReadParameter.bError THEN 
					// Execute with FALSE
					fbReadParameter(bExecute:= FALSE);
				END_IF
		END_IF
		
		// Diagnostic message present 
		stAxisStatus.bDiagMessage					:= stDriveStatus.nS135_DriveStatusWord.bS135_Class3_Diag_Mess;  
		// Warning message present 
		stAxisStatus.bWarning						:= stDriveStatus.nS135_DriveStatusWord.bS135_Class2_Diag_Warn;  
		// Error message present 
		stAxisStatus.bError							:= stDriveStatus.nS135_DriveStatusWord.bS135_Class1_Diag_Err;  
		// Diagnostic message number 
		{attribute 'displaymode':='hexadecimal'} 
		stAxisStatus.nDiagMessage					:= stDriveStatus.nS390_DiagnosticMessageNumber;
		
		// Display motion actual values 
		// Actual position (scale by 10000) 
		stAxisStatus.fActualPosition		:= DINT_TO_LREAL(stDriveStatus.nS386_ActivePositionFeedbackValue) / 10000.0; 
		// Actual velocity (scale by 1000) 
		stAxisStatus.fActualVelocity		:= DINT_TO_LREAL(stDriveStatus.nS40_VelocityFeedbackValue) / 1000.0; 
		// Actual Torque (scale by 10) 
		stAxisStatus.fActualTorque			:= INT_TO_LREAL(stDriveStatus.nS84_TorqueFeedback) / 10.0; 
		// Actual position error (scale by 10000) 
		stAxisStatus.fPositionError		:= DINT_TO_LREAL(stDriveStatus.nS189_PositionError) / 10000.0; 

(*==================================================================================================================================================
=============    COMMANDS TO THE DRIVE    ==========================================================================================================
==================================================================================================================================================*)
 	// Transfer and possibly scale command to the drive 
		// Operation mode 	
 		IF stAxisCommands.eOperationMode = E_OPERATION_MODE_NO.ePrimaryOpMode THEN 
			stDriveCommands.stS134_MasterControlWord.bS134_CmdOperationMode_Bit0 := FALSE;
			stDriveCommands.stS134_MasterControlWord.bS134_CmdOperationMode_Bit1 := FALSE;
			stDriveCommands.stS134_MasterControlWord.bS134_CmdOperationMode_Bit2 := FALSE;
		ELSIF stAxisCommands.eOperationMode = E_OPERATION_MODE_NO.eSecondaryOpMode1 THEN 
			stDriveCommands.stS134_MasterControlWord.bS134_CmdOperationMode_Bit0 := TRUE;
			stDriveCommands.stS134_MasterControlWord.bS134_CmdOperationMode_Bit1 := FALSE;
			stDriveCommands.stS134_MasterControlWord.bS134_CmdOperationMode_Bit2 := FALSE;
		ELSIF stAxisCommands.eOperationMode = E_OPERATION_MODE_NO.eSecondaryOpMode2 THEN 
			stDriveCommands.stS134_MasterControlWord.bS134_CmdOperationMode_Bit0 := FALSE;
			stDriveCommands.stS134_MasterControlWord.bS134_CmdOperationMode_Bit1 := TRUE;
			stDriveCommands.stS134_MasterControlWord.bS134_CmdOperationMode_Bit2 := FALSE;
		ELSIF stAxisCommands.eOperationMode = E_OPERATION_MODE_NO.eSecondaryOpMode3 THEN 
			stDriveCommands.stS134_MasterControlWord.bS134_CmdOperationMode_Bit0 := TRUE;
			stDriveCommands.stS134_MasterControlWord.bS134_CmdOperationMode_Bit1 := TRUE;
			stDriveCommands.stS134_MasterControlWord.bS134_CmdOperationMode_Bit2 := FALSE;
		ELSIF stAxisCommands.eOperationMode = E_OPERATION_MODE_NO.eSecondaryOpMode4 THEN 
			stDriveCommands.stS134_MasterControlWord.bS134_CmdOperationMode_Bit0 := FALSE;
			stDriveCommands.stS134_MasterControlWord.bS134_CmdOperationMode_Bit1 := FALSE;
			stDriveCommands.stS134_MasterControlWord.bS134_CmdOperationMode_Bit2 := TRUE;
		ELSIF stAxisCommands.eOperationMode = E_OPERATION_MODE_NO.eSecondaryOpMode5 THEN 
			stDriveCommands.stS134_MasterControlWord.bS134_CmdOperationMode_Bit0 := TRUE;
			stDriveCommands.stS134_MasterControlWord.bS134_CmdOperationMode_Bit1 := FALSE;
			stDriveCommands.stS134_MasterControlWord.bS134_CmdOperationMode_Bit2 := TRUE;
		ELSIF stAxisCommands.eOperationMode = E_OPERATION_MODE_NO.eSecondaryOpMode6 THEN 
			stDriveCommands.stS134_MasterControlWord.bS134_CmdOperationMode_Bit0 := FALSE;
			stDriveCommands.stS134_MasterControlWord.bS134_CmdOperationMode_Bit1 := TRUE;
			stDriveCommands.stS134_MasterControlWord.bS134_CmdOperationMode_Bit2 := TRUE;
		ELSIF stAxisCommands.eOperationMode = E_OPERATION_MODE_NO.eSecondaryOpMode7 THEN 
			stDriveCommands.stS134_MasterControlWord.bS134_CmdOperationMode_Bit0 := TRUE;
			stDriveCommands.stS134_MasterControlWord.bS134_CmdOperationMode_Bit1 := TRUE;
			stDriveCommands.stS134_MasterControlWord.bS134_CmdOperationMode_Bit2 := TRUE;
		END_IF
		
		// Enabling of the Axis 
		IF (NOT stAxisCommands.bEnableAxis) THEN 
			stDriveCommands.stS134_MasterControlWord.bS134_DriveEnable	:= TRUE; 
			stDriveCommands.stS134_MasterControlWord.bS134_DriveOn		:= FALSE; 
			stDriveCommands.stS134_MasterControlWord.bS134_DriveHalt	:= FALSE; 
		ELSIF stAxisCommands.bEnableAxis AND (NOT stAxisCommands.bHaltAxis) THEN 
			stDriveCommands.stS134_MasterControlWord.bS134_DriveEnable	:= TRUE; 
			stDriveCommands.stS134_MasterControlWord.bS134_DriveOn		:= TRUE; 
			stDriveCommands.stS134_MasterControlWord.bS134_DriveHalt	:= FALSE; 
		ELSIF stAxisCommands.bEnableAxis AND stAxisCommands.bHaltAxis THEN 
			stDriveCommands.stS134_MasterControlWord.bS134_DriveEnable	:= TRUE; 
			stDriveCommands.stS134_MasterControlWord.bS134_DriveOn		:= TRUE; 
			stDriveCommands.stS134_MasterControlWord.bS134_DriveHalt	:= TRUE; 
		END_IF
		
		// Positioning, Jog or stop the axis 
		CASE stAxisCommands.eMotionMode OF 
			E_MOTION_MODE.eStop: 
				stDriveCommands.stS145_SignalControlWord.bS346_1_PosCtrlWord_PosActivation	:= TRUE; 
				stDriveCommands.stS145_SignalControlWord.bS346_2_PosCtrlWord_PosActivation	:= TRUE; 				
			E_MOTION_MODE.eJogPositive: 
				stDriveCommands.stS145_SignalControlWord.bS346_1_PosCtrlWord_PosActivation	:= TRUE; 
				stDriveCommands.stS145_SignalControlWord.bS346_2_PosCtrlWord_PosActivation	:= FALSE; 				
			E_MOTION_MODE.eJogNegative: 
				stDriveCommands.stS145_SignalControlWord.bS346_1_PosCtrlWord_PosActivation	:= FALSE; 
				stDriveCommands.stS145_SignalControlWord.bS346_2_PosCtrlWord_PosActivation	:= TRUE; 				
			E_MOTION_MODE.ePositioning: 
				stDriveCommands.stS145_SignalControlWord.bS346_1_PosCtrlWord_PosActivation	:= FALSE; 
				stDriveCommands.stS145_SignalControlWord.bS346_2_PosCtrlWord_PosActivation	:= FALSE; 	
ii:=ii-1;			
		END_CASE
		
		// Position command change 
		stDriveCommands.stS145_SignalControlWord.bS346_5_PosCtrlWord_ImmBlockChange	:= stAxisCommands.bCommandPositionChange; 

		// Command position depending on Operation mode 
		IF stAxisStatus.nDiagMessage >= 16#C00A0102 AND stAxisStatus.nDiagMessage <= 16#C00A0105 THEN 
			stDriveCommands.nS47_PositionCommandValue 	:= LREAL_TO_DINT(10000.0 * stAxisCommands.fCommandPosition);
			stDriveCommands.nS282_PositioningCommandValue 	:= stDriveStatus.nS386_ActivePositionFeedbackValue;
			stDriveCommands.nS258_TargetPosition 		:= stDriveStatus.nS386_ActivePositionFeedbackValue;
		ELSIF (stAxisStatus.nDiagMessage >= 16#C00A0150 AND stAxisStatus.nDiagMessage <= 16#C00A0153) OR stAxisStatus.nDiagMessage = 16#C00A0161 THEN 
			stDriveCommands.nS282_PositioningCommandValue := LREAL_TO_DINT(10000.0 * stAxisCommands.fCommandPosition);
			stDriveCommands.nS47_PositionCommandValue 	:= stDriveStatus.nS386_ActivePositionFeedbackValue;
			stDriveCommands.nS258_TargetPosition 		:= stDriveStatus.nS386_ActivePositionFeedbackValue;
		ELSIF (stAxisStatus.nDiagMessage >= 16#C00A0106 AND stAxisStatus.nDiagMessage <= 16#C00A0109) THEN 
			stDriveCommands.nS258_TargetPosition := LREAL_TO_DINT(10000.0 * stAxisCommands.fCommandPosition);
			stDriveCommands.nS47_PositionCommandValue 	:= stDriveStatus.nS386_ActivePositionFeedbackValue;
			stDriveCommands.nS282_PositioningCommandValue 	:= stDriveStatus.nS386_ActivePositionFeedbackValue;
		END_IF
		
		// Target velocity 
		stDriveCommands.nS259_PositioningVelocity := LREAL_TO_UDINT(10000.0 * stAxisCommands.fCommandVelocity);
		
		// Target acceleration 
		stDriveCommands.nS260_PositioningAcceleration := LREAL_TO_UDINT(1000.0 * stAxisCommands.fCommandAcceleration);
		
		// Target deceleration 
		stDriveCommands.nS359_PositioningDeceleration := LREAL_TO_UDINT(1000.0 * stAxisCommands.fCommandDeceleration);

		// Feedrate override
		stDriveCommands.nS108_FeedrateOverride := LREAL_TO_UINT(100.0 * stAxisCommands.fFeedrateOverride);
		
		// Torque limit
		stDriveCommands.nS92_BiPolarTorqueLimit := LREAL_TO_INT(10.0 * stAxisCommands.fTorqueLimit);
		
		// Absolute or Relative target position values 
		stDriveCommands.stS145_SignalControlWord.bS346_3_PosCtrlWord_Abs_Rel := stAxisCommands.bPositionCommandValue;
		
		// Error reset 
		stDriveCommands.stS145_SignalControlWord.bS99_DriveErrorReset := stAxisCommands.bCmd_ErrorReset;
		
		// Set Absolute position 
		stDriveCommands.stS145_SignalControlWord.bP12_C300_SetAbsolutePosition := stAxisCommands.bCmd_SetAbsolutePosition;
		
		// Drive controlled homing
		stDriveCommands.stS145_SignalControlWord.bS148_C600_DriveControlledHoming := stAxisCommands.bCmd_DriveControlledHoming;

		// C1300 Disable monitoring command (in documentation called Positive Stop Drive Procedure) 
		stDriveCommands.stS145_SignalControlWord.bS159_C1300_Disable_Monitoring	:= stAxisCommands.bCmd_DisableLimits;

		// Activate parameter mode
		stDriveCommands.stS145_SignalControlWord.bS420_C0400_Activate_ParameterMode := stAxisCommands.bCmd_ActivateParameterMode;
		
		// Exit parameter mode
		stDriveCommands.stS145_SignalControlWord.bS422_C0200_Exit_ParameterMode := stAxisCommands.bCmd_ExitParameterMode;

		// Command value accept
		stDriveCommands.stS145_SignalControlWord.bS346_0_PosCtrlWord_CmdValueAccept := stAxisCommands.bCommandValueAccept; 
		
		stDriveCommands.nS40_VelocityCommandValue := LREAL_TO_UDINT(10000.0 * stAxisCommands.fVelocityCommandValue);

		// Run the Virtual Master
		IF stAxisCommands.bCmd_RunVirtualMater THEN 
			stDriveCommands.stS145_SignalControlWord.bP760_VM_PosCtrlWord_1_PosActivation	:= TRUE;
			stDriveCommands.stS145_SignalControlWord.bP760_VM_PosCtrlWord_2_PosActivation	:= FALSE;
			stDriveCommands.stS145_SignalControlWord.bP760_VM_PosCtrlWord_CmdValueAccept	:= TRUE;
		ELSE
			stDriveCommands.stS145_SignalControlWord.bP760_VM_PosCtrlWord_1_PosActivation	:= TRUE;
			stDriveCommands.stS145_SignalControlWord.bP760_VM_PosCtrlWord_2_PosActivation	:= TRUE;
			stDriveCommands.stS145_SignalControlWord.bP760_VM_PosCtrlWord_CmdValueAccept	:= FALSE;
		END_IF

END_FUNCTION_BLOCK
